/// calibration that is determined by calibration sequences of the unit (static offsets, shifts)
TYPE GearDataCalibration :
STRUCT
  OffsetRotationC : LREAL;
END_STRUCT
END_TYPE

(* stored: Version 1.1.0.1
   DUT GearDataCalibration: Id {7d0eb64c-7a40-47eb-b2a9-cbb61d9f9287} *)
